FUNCTION_BLOCK TC_OutputMapping (* Service Interface Function Block Type *)
  (* Standard: ISO 11783-6; Classification: Button – ISO 11783-6 – B.7; Function: All Outputs; Type: UT according to ISO 11783-6; Description: this maps to IX *)
  (* Version 1.0, 2018-12-05, Jose Cabral *)
  (* Version 1.1, 2022-08-04, Franz Höpfinger, HR Agrartechnik GmbH *)
  (* Version 1.2, 2023-01-05, Franz Höpfinger, HR Agrartechnik GmbH *)
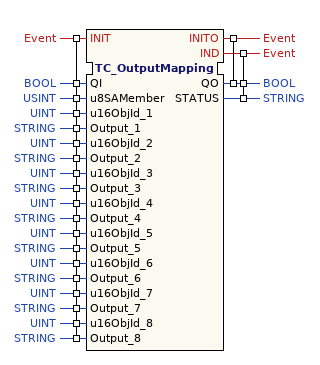
  EVENT_INPUT
    INIT WITH QI, u8SAMember, u16ObjId_1, Output_1, u16ObjId_2, Output_2, u16ObjId_3, Output_3, u16ObjId_4, Output_4, u16ObjId_5, Output_5, u16ObjId_6, Output_6, u16ObjId_7, Output_7, u16ObjId_8, Output_8; (* Service Initialization *)
  END_EVENT
  EVENT_OUTPUT
    INITO WITH QO; (* Initialization Confirm *)
    IND WITH QO, STATUS; (* Indication from Resource *)
  END_EVENT
  VAR_INPUT
    QI : BOOL; (* Event Output Qualifier *)
    u8SAMember : USINT := GLOBAL; (* Dummy !, set to GLOBAL if in doubt. OFF deactivates FB. *)
    u16ObjId_1 : UINT; (* Object ID of Output 1 *)
    Output_1 : STRING; (* Identifier for Output 1 *)
    u16ObjId_2 : UINT; (* Object ID of Output 2 *)
    Output_2 : STRING; (* Identifier for Output 2 *)
    u16ObjId_3 : UINT; (* Object ID of Output 3 *)
    Output_3 : STRING; (* Identifier for Output 3 *)
    u16ObjId_4 : UINT; (* Object ID of Output 4 *)
    Output_4 : STRING; (* Identifier for Output 4 *)
    u16ObjId_5 : UINT; (* Object ID of Output 5 *)
    Output_5 : STRING; (* Identifier for Output 5 *)
    u16ObjId_6 : UINT; (* Object ID of Output 6 *)
    Output_6 : STRING; (* Identifier for Output 6 *)
    u16ObjId_7 : UINT; (* Object ID of Output 7 *)
    Output_7 : STRING; (* Identifier for Output 7 *)
    u16ObjId_8 : UINT; (* Object ID of Output 8 *)
    Output_8 : STRING; (* Identifier for Output 8 *)
  END_VAR
  VAR_OUTPUT
    QO : BOOL; (* Event Output Qualifier *)
    STATUS : STRING; (* Service Status *)
  END_VAR
END_FUNCTION_BLOCK
